// TIA Portal V17 export
// export: Created 2026-07-06T15:33:03.9431546Z, ExportSetting WithDefaults, DisplayName Totally Integrated Automation Portal, DisplayVersion V17, DisplayName TIA Portal Openness, DisplayVersion V17, DisplayName TIA Portal Version Control Interface, DisplayVersion V17, DisplayName STEP 7 Professional, DisplayVersion V17, DisplayName STEP 7 Safety, DisplayVersion V17, DisplayName WinCC Professional, DisplayVersion V17
DATA_BLOCK "Canet_com_DB"   // DB20
VERSION : 0.1
// stored: AutoNumber true, DBAccessibleFromOPCUA true, InstanceOfName Canet_com, InstanceOfType FB
"Canet_com"
   // VAR_INPUT
   //    con_req : Bool;
   // END_VAR
   // VAR_OUTPUT
   //    connection_established : Bool;
   // END_VAR
   // VAR_IN_OUT
   //    Data_rcvd : Array[0..12] of Byte;
   // END_VAR
BEGIN
END_DATA_BLOCK
